// TIA Portal V20 export
DATA_BLOCK "LBP_CtrlEnergy"   // DB1000
TITLE = Ctrl-Energy
{ S7_Optimized_Access := 'FALSE'; DB_Accessible_From_OPC_UA := 'FALSE' }
AUTHOR : SINUMERIK
FAMILY : SINUMERIK_ONE
VERSION : 6.24
// Interface between user program and operating software, contains energy-saving profiles for Ctrl-Energy / Interface entre programme utilisateur et logiciel d'exploitation contient des profils d'économie d'énergie pour Ctrl-Energy
// stored: AutoNumber false, DBAccessibleFromOPCUA false, DBAccessibleFromWebserver false
   VAR RETAIN
      Profile : Array[1..8] of Struct
         ESaveOn { ExternalWritable := 'False'} : Bool;   // Activate energy-saving profile immediately / Activer immédiatement le profil d'économie d'énergie
         ReloadT2 { ExternalWritable := 'False'} : Bool;   // Reload Prewarning time (T2) / Recharger temps de préavis (T2)
         res0_2 { ExternalWritable := 'False'} : Bool;
         res0_3 { ExternalWritable := 'False'} : Bool;
         res0_4 { ExternalWritable := 'False'} : Bool;
         res0_5 { ExternalWritable := 'False'} : Bool;
         res0_6 { ExternalWritable := 'False'} : Bool;
         res0_7 { ExternalWritable := 'False'} : Bool;
         HmiESaveOn : Bool;   // HMI->PLC: Activate energy-saving profile immediately / IHM->AP : activer immédiatement le profil d'économie d'énergie
         res1_1 { ExternalWritable := 'False'} : Bool;
         res1_2 { ExternalWritable := 'False'} : Bool;
         res1_3 { ExternalWritable := 'False'} : Bool;
         res1_4 { ExternalWritable := 'False'} : Bool;
         res1_5 { ExternalWritable := 'False'} : Bool;
         res1_6 { ExternalWritable := 'False'} : Bool;
         res1_7 { ExternalWritable := 'False'} : Bool;
         MasterCompSig { ExternalWritable := 'False'} : Bool;   // Master computer signal / Signal ordinateur maître
         PlcUserSig { ExternalWritable := 'False'} : Bool;   // PLC user signal / AP signal utilisateur
         res2_2 { ExternalWritable := 'False'} : Bool;
         res2_3 { ExternalWritable := 'False'} : Bool;
         res2_4 { ExternalWritable := 'False'} : Bool;
         res2_5 { ExternalWritable := 'False'} : Bool;
         res2_6 { ExternalWritable := 'False'} : Bool;
         res2_7 { ExternalWritable := 'False'} : Bool;
         res3 { ExternalWritable := 'False'} : Byte;
         ESaveIsOn { ExternalWritable := 'False'} : Bool;   // Energy-saving state active / État économie d'énergie actif
         T1Expired { ExternalWritable := 'False'} : Bool;   // Activation time T1 expired / Temps d'activation T1 écoulé
         res4_2 { ExternalWritable := 'False'} : Bool;
         res4_3 { ExternalWritable := 'False'} : Bool;
         res4_4 { ExternalWritable := 'False'} : Bool;
         res4_5 { ExternalWritable := 'False'} : Bool;
         res4_6 { ExternalWritable := 'False'} : Bool;
         res4_7 { ExternalWritable := 'False'} : Bool;
         res5 { ExternalWritable := 'False'} : Byte;
         ActValT1 { ExternalWritable := 'False'} : Int;   // T1 current value / T1 valeur réelle
         ActValT2 { ExternalWritable := 'False'} : Int;   // T2 current value / T2 valeur réelle
         ESaveValid : Bool;   // HMI->PLC: Energy-saving profile valid / IHM->AP : profil d'économie d'énergie valide
         ESaveOff : Bool;   // HMI->PLC: Deactivate energy-saving profileblock energy-saving profile / IHM->AP : désactiver/bloquer le profil d'économie d'énergie
         res10_2 { ExternalWritable := 'False'} : Bool;
         res10_3 { ExternalWritable := 'False'} : Bool;
         res10_4 { ExternalWritable := 'False'} : Bool;
         res10_5 { ExternalWritable := 'False'} : Bool;
         res10_6 { ExternalWritable := 'False'} : Bool;
         res10_7 { ExternalWritable := 'False'} : Bool;
         CondOpPanel : Bool;   // HMI->PLC: Operator panel / IHM->AP : pupitre opérateur
         CondDataTransfer : Bool;   // HMI->PLC: Data transfer / IHM->AP : transmission de données
         CondWindowChange : Bool;   // HMI->PLC: Window change / IHM->AP : changement de fenêtre
         res11_3 { ExternalWritable := 'False'} : Bool;
         res11_4 { ExternalWritable := 'False'} : Bool;
         res11_5 { ExternalWritable := 'False'} : Bool;
         res11_6 { ExternalWritable := 'False'} : Bool;
         res11_7 { ExternalWritable := 'False'} : Bool;
         CondMCP : Bool;   // HMI->PLC: Machine control panel / IHM->AP : pupitre opérateur machine
         res12_1 { ExternalWritable := 'False'} : Bool;
         res12_2 { ExternalWritable := 'False'} : Bool;
         res12_3 { ExternalWritable := 'False'} : Bool;
         res12_4 { ExternalWritable := 'False'} : Bool;
         res12_5 { ExternalWritable := 'False'} : Bool;
         res12_6 { ExternalWritable := 'False'} : Bool;
         res12_7 { ExternalWritable := 'False'} : Bool;
         CondNcChan1 : Bool;   // HMI->PLC: NC channel 1 in reset / IHM->AP : canal CN 1 en Reset
         CondNcChan2 : Bool;   // HMI->PLC: NC channel 2 in reset / IHM->AP : canal CN 2 en Reset
         CondNcChan3 : Bool;   // HMI->PLC: NC channel 3 in reset / IHM->AP : canal CN 3 en Reset
         CondNcChan4 : Bool;   // HMI->PLC: NC channel 4 in reset / IHM->AP : canal CN 4 en Reset
         CondNcChan5 : Bool;   // HMI->PLC: NC channel 5 in reset / IHM->AP : canal CN 5 en Reset
         CondNcChan6 : Bool;   // HMI->PLC: NC channel 6 in reset / IHM->AP : canal CN 6 en Reset
         CondNcChan7 : Bool;   // HMI->PLC: NC channel 7 in reset / IHM->AP : canal CN 7 en Reset
         CondNcChan8 : Bool;   // HMI->PLC: NC channel 8 in reset / IHM->AP : canal CN 8 en Reset
         CondNcChan9 : Bool;   // HMI->PLC: NC channel 9 in reset / IHM->AP : canal CN 9 en Reset
         CondNcChan10 : Bool;   // HMI->PLC: NC channel 10 in reset / IHM->AP : canal CN 10 en Reset
         res14_2 { ExternalWritable := 'False'} : Bool;
         res14_3 { ExternalWritable := 'False'} : Bool;
         res14_4 { ExternalWritable := 'False'} : Bool;
         res14_5 { ExternalWritable := 'False'} : Bool;
         res14_6 { ExternalWritable := 'False'} : Bool;
         res14_7 { ExternalWritable := 'False'} : Bool;
         CondMasterCompSig : Bool;   // HMI->PLC: Master computer signal / IHM->AP : signal ordinateur maître
         CondPlcUserSig : Bool;   // HMI->PLC: PLC user signal / IHM->AP : signal utilisateur AP
         res15_2 { ExternalWritable := 'False'} : Bool;
         res15_3 { ExternalWritable := 'False'} : Bool;
         res15_4 { ExternalWritable := 'False'} : Bool;
         res15_5 { ExternalWritable := 'False'} : Bool;
         res15_6 { ExternalWritable := 'False'} : Bool;
         res15_7 { ExternalWritable := 'False'} : Bool;
         PresetT1 : Int;   // HMI->PLC: Activation time T1 / IHM->AP : temps d'activation T1
         PresetT2 : Int;   // HMI->PLC: Prewarning time T2 / IHM->AP : temps de préavis T2
      END_STRUCT;
   END_VAR
BEGIN
   // Profile[2].ESaveOn : Activate energy-saving profile immediately / Activer immédiatement le profil d'économie d'énergie
   // Profile[3].ESaveOn : Activate energy-saving profile immediately / Activer immédiatement le profil d'économie d'énergie
   // Profile[4].ESaveOn : Activate energy-saving profile immediately / Activer immédiatement le profil d'économie d'énergie
   // Profile[5].ESaveOn : Activate energy-saving profile immediately / Activer immédiatement le profil d'économie d'énergie
   // Profile[6].ESaveOn : Activate energy-saving profile immediately / Activer immédiatement le profil d'économie d'énergie
   // Profile[7].ESaveOn : Activate energy-saving profile immediately / Activer immédiatement le profil d'économie d'énergie
   // Profile[8].ESaveOn : Activate energy-saving profile immediately / Activer immédiatement le profil d'économie d'énergie
   // Profile[2].ReloadT2 : Reload Prewarning time (T2) / Recharger temps de préavis (T2)
   // Profile[3].ReloadT2 : Reload Prewarning time (T2) / Recharger temps de préavis (T2)
   // Profile[4].ReloadT2 : Reload Prewarning time (T2) / Recharger temps de préavis (T2)
   // Profile[5].ReloadT2 : Reload Prewarning time (T2) / Recharger temps de préavis (T2)
   // Profile[6].ReloadT2 : Reload Prewarning time (T2) / Recharger temps de préavis (T2)
   // Profile[7].ReloadT2 : Reload Prewarning time (T2) / Recharger temps de préavis (T2)
   // Profile[8].ReloadT2 : Reload Prewarning time (T2) / Recharger temps de préavis (T2)
   // Profile[2].HmiESaveOn : HMI->PLC: Activate energy-saving profile immediately / IHM->AP : activer immédiatement le profil d'économie d'énergie
   // Profile[3].HmiESaveOn : HMI->PLC: Activate energy-saving profile immediately / IHM->AP : activer immédiatement le profil d'économie d'énergie
   // Profile[4].HmiESaveOn : HMI->PLC: Activate energy-saving profile immediately / IHM->AP : activer immédiatement le profil d'économie d'énergie
   // Profile[5].HmiESaveOn : HMI->PLC: Activate energy-saving profile immediately / IHM->AP : activer immédiatement le profil d'économie d'énergie
   // Profile[6].HmiESaveOn : HMI->PLC: Activate energy-saving profile immediately / IHM->AP : activer immédiatement le profil d'économie d'énergie
   // Profile[7].HmiESaveOn : HMI->PLC: Activate energy-saving profile immediately / IHM->AP : activer immédiatement le profil d'économie d'énergie
   // Profile[8].HmiESaveOn : HMI->PLC: Activate energy-saving profile immediately / IHM->AP : activer immédiatement le profil d'économie d'énergie
   // Profile[2].MasterCompSig : Master computer signal / Signal ordinateur maître
   // Profile[3].MasterCompSig : Master computer signal / Signal ordinateur maître
   // Profile[4].MasterCompSig : Master computer signal / Signal ordinateur maître
   // Profile[5].MasterCompSig : Master computer signal / Signal ordinateur maître
   // Profile[6].MasterCompSig : Master computer signal / Signal ordinateur maître
   // Profile[7].MasterCompSig : Master computer signal / Signal ordinateur maître
   // Profile[8].MasterCompSig : Master computer signal / Signal ordinateur maître
   // Profile[2].PlcUserSig : PLC user signal / AP signal utilisateur
   // Profile[3].PlcUserSig : PLC user signal / AP signal utilisateur
   // Profile[4].PlcUserSig : PLC user signal / AP signal utilisateur
   // Profile[5].PlcUserSig : PLC user signal / AP signal utilisateur
   // Profile[6].PlcUserSig : PLC user signal / AP signal utilisateur
   // Profile[7].PlcUserSig : PLC user signal / AP signal utilisateur
   // Profile[8].PlcUserSig : PLC user signal / AP signal utilisateur
   // Profile[2].ESaveIsOn : Energy-saving state active / État économie d'énergie actif
   // Profile[3].ESaveIsOn : Energy-saving state active / État économie d'énergie actif
   // Profile[4].ESaveIsOn : Energy-saving state active / État économie d'énergie actif
   // Profile[5].ESaveIsOn : Energy-saving state active / État économie d'énergie actif
   // Profile[6].ESaveIsOn : Energy-saving state active / État économie d'énergie actif
   // Profile[7].ESaveIsOn : Energy-saving state active / État économie d'énergie actif
   // Profile[8].ESaveIsOn : Energy-saving state active / État économie d'énergie actif
   // Profile[2].T1Expired : Activation time T1 expired / Temps d'activation T1 écoulé
   // Profile[3].T1Expired : Activation time T1 expired / Temps d'activation T1 écoulé
   // Profile[4].T1Expired : Activation time T1 expired / Temps d'activation T1 écoulé
   // Profile[5].T1Expired : Activation time T1 expired / Temps d'activation T1 écoulé
   // Profile[6].T1Expired : Activation time T1 expired / Temps d'activation T1 écoulé
   // Profile[7].T1Expired : Activation time T1 expired / Temps d'activation T1 écoulé
   // Profile[8].T1Expired : Activation time T1 expired / Temps d'activation T1 écoulé
   // Profile[2].ActValT1 : T1 current value / T1 valeur réelle
   // Profile[3].ActValT1 : T1 current value / T1 valeur réelle
   // Profile[4].ActValT1 : T1 current value / T1 valeur réelle
   // Profile[5].ActValT1 : T1 current value / T1 valeur réelle
   // Profile[6].ActValT1 : T1 current value / T1 valeur réelle
   // Profile[7].ActValT1 : T1 current value / T1 valeur réelle
   // Profile[8].ActValT1 : T1 current value / T1 valeur réelle
   // Profile[2].ActValT2 : T2 current value / T2 valeur réelle
   // Profile[3].ActValT2 : T2 current value / T2 valeur réelle
   // Profile[4].ActValT2 : T2 current value / T2 valeur réelle
   // Profile[5].ActValT2 : T2 current value / T2 valeur réelle
   // Profile[6].ActValT2 : T2 current value / T2 valeur réelle
   // Profile[7].ActValT2 : T2 current value / T2 valeur réelle
   // Profile[8].ActValT2 : T2 current value / T2 valeur réelle
   Profile[1].ESaveValid := TRUE;
   Profile[2].ESaveValid := TRUE;   // HMI->PLC: Energy-saving profile valid / IHM->AP : profil d'économie d'énergie valide
   Profile[3].ESaveValid := TRUE;   // HMI->PLC: Energy-saving profile valid / IHM->AP : profil d'économie d'énergie valide
   // Profile[4].ESaveValid : HMI->PLC: Energy-saving profile valid / IHM->AP : profil d'économie d'énergie valide
   // Profile[5].ESaveValid : HMI->PLC: Energy-saving profile valid / IHM->AP : profil d'économie d'énergie valide
   // Profile[6].ESaveValid : HMI->PLC: Energy-saving profile valid / IHM->AP : profil d'économie d'énergie valide
   // Profile[7].ESaveValid : HMI->PLC: Energy-saving profile valid / IHM->AP : profil d'économie d'énergie valide
   // Profile[8].ESaveValid : HMI->PLC: Energy-saving profile valid / IHM->AP : profil d'économie d'énergie valide
   Profile[1].ESaveOff := TRUE;
   Profile[2].ESaveOff := TRUE;   // HMI->PLC: Deactivate energy-saving profileblock energy-saving profile / IHM->AP : désactiver/bloquer le profil d'économie d'énergie
   Profile[3].ESaveOff := TRUE;   // HMI->PLC: Deactivate energy-saving profileblock energy-saving profile / IHM->AP : désactiver/bloquer le profil d'économie d'énergie
   // Profile[4].ESaveOff : HMI->PLC: Deactivate energy-saving profileblock energy-saving profile / IHM->AP : désactiver/bloquer le profil d'économie d'énergie
   // Profile[5].ESaveOff : HMI->PLC: Deactivate energy-saving profileblock energy-saving profile / IHM->AP : désactiver/bloquer le profil d'économie d'énergie
   // Profile[6].ESaveOff : HMI->PLC: Deactivate energy-saving profileblock energy-saving profile / IHM->AP : désactiver/bloquer le profil d'économie d'énergie
   // Profile[7].ESaveOff : HMI->PLC: Deactivate energy-saving profileblock energy-saving profile / IHM->AP : désactiver/bloquer le profil d'économie d'énergie
   // Profile[8].ESaveOff : HMI->PLC: Deactivate energy-saving profileblock energy-saving profile / IHM->AP : désactiver/bloquer le profil d'économie d'énergie
   // Profile[2].CondOpPanel : HMI->PLC: Operator panel / IHM->AP : pupitre opérateur
   Profile[3].CondOpPanel := TRUE;   // HMI->PLC: Operator panel / IHM->AP : pupitre opérateur
   // Profile[4].CondOpPanel : HMI->PLC: Operator panel / IHM->AP : pupitre opérateur
   // Profile[5].CondOpPanel : HMI->PLC: Operator panel / IHM->AP : pupitre opérateur
   // Profile[6].CondOpPanel : HMI->PLC: Operator panel / IHM->AP : pupitre opérateur
   // Profile[7].CondOpPanel : HMI->PLC: Operator panel / IHM->AP : pupitre opérateur
   // Profile[8].CondOpPanel : HMI->PLC: Operator panel / IHM->AP : pupitre opérateur
   // Profile[2].CondDataTransfer : HMI->PLC: Data transfer / IHM->AP : transmission de données
   Profile[3].CondDataTransfer := TRUE;   // HMI->PLC: Data transfer / IHM->AP : transmission de données
   // Profile[4].CondDataTransfer : HMI->PLC: Data transfer / IHM->AP : transmission de données
   // Profile[5].CondDataTransfer : HMI->PLC: Data transfer / IHM->AP : transmission de données
   // Profile[6].CondDataTransfer : HMI->PLC: Data transfer / IHM->AP : transmission de données
   // Profile[7].CondDataTransfer : HMI->PLC: Data transfer / IHM->AP : transmission de données
   // Profile[8].CondDataTransfer : HMI->PLC: Data transfer / IHM->AP : transmission de données
   // Profile[2].CondWindowChange : HMI->PLC: Window change / IHM->AP : changement de fenêtre
   Profile[3].CondWindowChange := TRUE;   // HMI->PLC: Window change / IHM->AP : changement de fenêtre
   // Profile[4].CondWindowChange : HMI->PLC: Window change / IHM->AP : changement de fenêtre
   // Profile[5].CondWindowChange : HMI->PLC: Window change / IHM->AP : changement de fenêtre
   // Profile[6].CondWindowChange : HMI->PLC: Window change / IHM->AP : changement de fenêtre
   // Profile[7].CondWindowChange : HMI->PLC: Window change / IHM->AP : changement de fenêtre
   // Profile[8].CondWindowChange : HMI->PLC: Window change / IHM->AP : changement de fenêtre
   Profile[2].CondMCP := TRUE;   // HMI->PLC: Machine control panel / IHM->AP : pupitre opérateur machine
   Profile[3].CondMCP := TRUE;   // HMI->PLC: Machine control panel / IHM->AP : pupitre opérateur machine
   // Profile[4].CondMCP : HMI->PLC: Machine control panel / IHM->AP : pupitre opérateur machine
   // Profile[5].CondMCP : HMI->PLC: Machine control panel / IHM->AP : pupitre opérateur machine
   // Profile[6].CondMCP : HMI->PLC: Machine control panel / IHM->AP : pupitre opérateur machine
   // Profile[7].CondMCP : HMI->PLC: Machine control panel / IHM->AP : pupitre opérateur machine
   // Profile[8].CondMCP : HMI->PLC: Machine control panel / IHM->AP : pupitre opérateur machine
   Profile[1].CondNcChan1 := TRUE;
   Profile[2].CondNcChan1 := TRUE;   // HMI->PLC: NC channel 1 in reset / IHM->AP : canal CN 1 en Reset
   Profile[3].CondNcChan1 := TRUE;   // HMI->PLC: NC channel 1 in reset / IHM->AP : canal CN 1 en Reset
   // Profile[4].CondNcChan1 : HMI->PLC: NC channel 1 in reset / IHM->AP : canal CN 1 en Reset
   // Profile[5].CondNcChan1 : HMI->PLC: NC channel 1 in reset / IHM->AP : canal CN 1 en Reset
   // Profile[6].CondNcChan1 : HMI->PLC: NC channel 1 in reset / IHM->AP : canal CN 1 en Reset
   // Profile[7].CondNcChan1 : HMI->PLC: NC channel 1 in reset / IHM->AP : canal CN 1 en Reset
   // Profile[8].CondNcChan1 : HMI->PLC: NC channel 1 in reset / IHM->AP : canal CN 1 en Reset
   Profile[1].CondNcChan2 := TRUE;
   Profile[2].CondNcChan2 := TRUE;   // HMI->PLC: NC channel 2 in reset / IHM->AP : canal CN 2 en Reset
   Profile[3].CondNcChan2 := TRUE;   // HMI->PLC: NC channel 2 in reset / IHM->AP : canal CN 2 en Reset
   // Profile[4].CondNcChan2 : HMI->PLC: NC channel 2 in reset / IHM->AP : canal CN 2 en Reset
   // Profile[5].CondNcChan2 : HMI->PLC: NC channel 2 in reset / IHM->AP : canal CN 2 en Reset
   // Profile[6].CondNcChan2 : HMI->PLC: NC channel 2 in reset / IHM->AP : canal CN 2 en Reset
   // Profile[7].CondNcChan2 : HMI->PLC: NC channel 2 in reset / IHM->AP : canal CN 2 en Reset
   // Profile[8].CondNcChan2 : HMI->PLC: NC channel 2 in reset / IHM->AP : canal CN 2 en Reset
   Profile[1].CondNcChan3 := TRUE;
   Profile[2].CondNcChan3 := TRUE;   // HMI->PLC: NC channel 3 in reset / IHM->AP : canal CN 3 en Reset
   Profile[3].CondNcChan3 := TRUE;   // HMI->PLC: NC channel 3 in reset / IHM->AP : canal CN 3 en Reset
   // Profile[4].CondNcChan3 : HMI->PLC: NC channel 3 in reset / IHM->AP : canal CN 3 en Reset
   // Profile[5].CondNcChan3 : HMI->PLC: NC channel 3 in reset / IHM->AP : canal CN 3 en Reset
   // Profile[6].CondNcChan3 : HMI->PLC: NC channel 3 in reset / IHM->AP : canal CN 3 en Reset
   // Profile[7].CondNcChan3 : HMI->PLC: NC channel 3 in reset / IHM->AP : canal CN 3 en Reset
   // Profile[8].CondNcChan3 : HMI->PLC: NC channel 3 in reset / IHM->AP : canal CN 3 en Reset
   Profile[1].CondNcChan4 := TRUE;
   Profile[2].CondNcChan4 := TRUE;   // HMI->PLC: NC channel 4 in reset / IHM->AP : canal CN 4 en Reset
   Profile[3].CondNcChan4 := TRUE;   // HMI->PLC: NC channel 4 in reset / IHM->AP : canal CN 4 en Reset
   // Profile[4].CondNcChan4 : HMI->PLC: NC channel 4 in reset / IHM->AP : canal CN 4 en Reset
   // Profile[5].CondNcChan4 : HMI->PLC: NC channel 4 in reset / IHM->AP : canal CN 4 en Reset
   // Profile[6].CondNcChan4 : HMI->PLC: NC channel 4 in reset / IHM->AP : canal CN 4 en Reset
   // Profile[7].CondNcChan4 : HMI->PLC: NC channel 4 in reset / IHM->AP : canal CN 4 en Reset
   // Profile[8].CondNcChan4 : HMI->PLC: NC channel 4 in reset / IHM->AP : canal CN 4 en Reset
   Profile[1].CondNcChan5 := TRUE;
   Profile[2].CondNcChan5 := TRUE;   // HMI->PLC: NC channel 5 in reset / IHM->AP : canal CN 5 en Reset
   Profile[3].CondNcChan5 := TRUE;   // HMI->PLC: NC channel 5 in reset / IHM->AP : canal CN 5 en Reset
   // Profile[4].CondNcChan5 : HMI->PLC: NC channel 5 in reset / IHM->AP : canal CN 5 en Reset
   // Profile[5].CondNcChan5 : HMI->PLC: NC channel 5 in reset / IHM->AP : canal CN 5 en Reset
   // Profile[6].CondNcChan5 : HMI->PLC: NC channel 5 in reset / IHM->AP : canal CN 5 en Reset
   // Profile[7].CondNcChan5 : HMI->PLC: NC channel 5 in reset / IHM->AP : canal CN 5 en Reset
   // Profile[8].CondNcChan5 : HMI->PLC: NC channel 5 in reset / IHM->AP : canal CN 5 en Reset
   Profile[1].CondNcChan6 := TRUE;
   Profile[2].CondNcChan6 := TRUE;   // HMI->PLC: NC channel 6 in reset / IHM->AP : canal CN 6 en Reset
   Profile[3].CondNcChan6 := TRUE;   // HMI->PLC: NC channel 6 in reset / IHM->AP : canal CN 6 en Reset
   // Profile[4].CondNcChan6 : HMI->PLC: NC channel 6 in reset / IHM->AP : canal CN 6 en Reset
   // Profile[5].CondNcChan6 : HMI->PLC: NC channel 6 in reset / IHM->AP : canal CN 6 en Reset
   // Profile[6].CondNcChan6 : HMI->PLC: NC channel 6 in reset / IHM->AP : canal CN 6 en Reset
   // Profile[7].CondNcChan6 : HMI->PLC: NC channel 6 in reset / IHM->AP : canal CN 6 en Reset
   // Profile[8].CondNcChan6 : HMI->PLC: NC channel 6 in reset / IHM->AP : canal CN 6 en Reset
   Profile[1].CondNcChan7 := TRUE;
   Profile[2].CondNcChan7 := TRUE;   // HMI->PLC: NC channel 7 in reset / IHM->AP : canal CN 7 en Reset
   Profile[3].CondNcChan7 := TRUE;   // HMI->PLC: NC channel 7 in reset / IHM->AP : canal CN 7 en Reset
   // Profile[4].CondNcChan7 : HMI->PLC: NC channel 7 in reset / IHM->AP : canal CN 7 en Reset
   // Profile[5].CondNcChan7 : HMI->PLC: NC channel 7 in reset / IHM->AP : canal CN 7 en Reset
   // Profile[6].CondNcChan7 : HMI->PLC: NC channel 7 in reset / IHM->AP : canal CN 7 en Reset
   // Profile[7].CondNcChan7 : HMI->PLC: NC channel 7 in reset / IHM->AP : canal CN 7 en Reset
   // Profile[8].CondNcChan7 : HMI->PLC: NC channel 7 in reset / IHM->AP : canal CN 7 en Reset
   Profile[1].CondNcChan8 := TRUE;
   Profile[2].CondNcChan8 := TRUE;   // HMI->PLC: NC channel 8 in reset / IHM->AP : canal CN 8 en Reset
   Profile[3].CondNcChan8 := TRUE;   // HMI->PLC: NC channel 8 in reset / IHM->AP : canal CN 8 en Reset
   // Profile[4].CondNcChan8 : HMI->PLC: NC channel 8 in reset / IHM->AP : canal CN 8 en Reset
   // Profile[5].CondNcChan8 : HMI->PLC: NC channel 8 in reset / IHM->AP : canal CN 8 en Reset
   // Profile[6].CondNcChan8 : HMI->PLC: NC channel 8 in reset / IHM->AP : canal CN 8 en Reset
   // Profile[7].CondNcChan8 : HMI->PLC: NC channel 8 in reset / IHM->AP : canal CN 8 en Reset
   // Profile[8].CondNcChan8 : HMI->PLC: NC channel 8 in reset / IHM->AP : canal CN 8 en Reset
   Profile[1].CondNcChan9 := TRUE;
   Profile[2].CondNcChan9 := TRUE;   // HMI->PLC: NC channel 9 in reset / IHM->AP : canal CN 9 en Reset
   Profile[3].CondNcChan9 := TRUE;   // HMI->PLC: NC channel 9 in reset / IHM->AP : canal CN 9 en Reset
   // Profile[4].CondNcChan9 : HMI->PLC: NC channel 9 in reset / IHM->AP : canal CN 9 en Reset
   // Profile[5].CondNcChan9 : HMI->PLC: NC channel 9 in reset / IHM->AP : canal CN 9 en Reset
   // Profile[6].CondNcChan9 : HMI->PLC: NC channel 9 in reset / IHM->AP : canal CN 9 en Reset
   // Profile[7].CondNcChan9 : HMI->PLC: NC channel 9 in reset / IHM->AP : canal CN 9 en Reset
   // Profile[8].CondNcChan9 : HMI->PLC: NC channel 9 in reset / IHM->AP : canal CN 9 en Reset
   Profile[1].CondNcChan10 := TRUE;
   Profile[2].CondNcChan10 := TRUE;   // HMI->PLC: NC channel 10 in reset / IHM->AP : canal CN 10 en Reset
   Profile[3].CondNcChan10 := TRUE;   // HMI->PLC: NC channel 10 in reset / IHM->AP : canal CN 10 en Reset
   // Profile[4].CondNcChan10 : HMI->PLC: NC channel 10 in reset / IHM->AP : canal CN 10 en Reset
   // Profile[5].CondNcChan10 : HMI->PLC: NC channel 10 in reset / IHM->AP : canal CN 10 en Reset
   // Profile[6].CondNcChan10 : HMI->PLC: NC channel 10 in reset / IHM->AP : canal CN 10 en Reset
   // Profile[7].CondNcChan10 : HMI->PLC: NC channel 10 in reset / IHM->AP : canal CN 10 en Reset
   // Profile[8].CondNcChan10 : HMI->PLC: NC channel 10 in reset / IHM->AP : canal CN 10 en Reset
   // Profile[2].CondMasterCompSig : HMI->PLC: Master computer signal / IHM->AP : signal ordinateur maître
   // Profile[3].CondMasterCompSig : HMI->PLC: Master computer signal / IHM->AP : signal ordinateur maître
   // Profile[4].CondMasterCompSig : HMI->PLC: Master computer signal / IHM->AP : signal ordinateur maître
   // Profile[5].CondMasterCompSig : HMI->PLC: Master computer signal / IHM->AP : signal ordinateur maître
   // Profile[6].CondMasterCompSig : HMI->PLC: Master computer signal / IHM->AP : signal ordinateur maître
   // Profile[7].CondMasterCompSig : HMI->PLC: Master computer signal / IHM->AP : signal ordinateur maître
   // Profile[8].CondMasterCompSig : HMI->PLC: Master computer signal / IHM->AP : signal ordinateur maître
   Profile[1].CondPlcUserSig := TRUE;
   Profile[2].CondPlcUserSig := TRUE;   // HMI->PLC: PLC user signal / IHM->AP : signal utilisateur AP
   Profile[3].CondPlcUserSig := TRUE;   // HMI->PLC: PLC user signal / IHM->AP : signal utilisateur AP
   // Profile[4].CondPlcUserSig : HMI->PLC: PLC user signal / IHM->AP : signal utilisateur AP
   // Profile[5].CondPlcUserSig : HMI->PLC: PLC user signal / IHM->AP : signal utilisateur AP
   // Profile[6].CondPlcUserSig : HMI->PLC: PLC user signal / IHM->AP : signal utilisateur AP
   // Profile[7].CondPlcUserSig : HMI->PLC: PLC user signal / IHM->AP : signal utilisateur AP
   // Profile[8].CondPlcUserSig : HMI->PLC: PLC user signal / IHM->AP : signal utilisateur AP
   Profile[1].PresetT1 := 60;
   Profile[2].PresetT1 := 120;   // HMI->PLC: Activation time T1 / IHM->AP : temps d'activation T1
   Profile[3].PresetT1 := 600;   // HMI->PLC: Activation time T1 / IHM->AP : temps d'activation T1
   // Profile[4].PresetT1 : HMI->PLC: Activation time T1 / IHM->AP : temps d'activation T1
   // Profile[5].PresetT1 : HMI->PLC: Activation time T1 / IHM->AP : temps d'activation T1
   // Profile[6].PresetT1 : HMI->PLC: Activation time T1 / IHM->AP : temps d'activation T1
   // Profile[7].PresetT1 : HMI->PLC: Activation time T1 / IHM->AP : temps d'activation T1
   // Profile[8].PresetT1 : HMI->PLC: Activation time T1 / IHM->AP : temps d'activation T1
   Profile[1].PresetT2 := 120;
   Profile[2].PresetT2 := 300;   // HMI->PLC: Prewarning time T2 / IHM->AP : temps de préavis T2
   // Profile[3].PresetT2 : HMI->PLC: Prewarning time T2 / IHM->AP : temps de préavis T2
   // Profile[4].PresetT2 : HMI->PLC: Prewarning time T2 / IHM->AP : temps de préavis T2
   // Profile[5].PresetT2 : HMI->PLC: Prewarning time T2 / IHM->AP : temps de préavis T2
   // Profile[6].PresetT2 : HMI->PLC: Prewarning time T2 / IHM->AP : temps de préavis T2
   // Profile[7].PresetT2 : HMI->PLC: Prewarning time T2 / IHM->AP : temps de préavis T2
   // Profile[8].PresetT2 : HMI->PLC: Prewarning time T2 / IHM->AP : temps de préavis T2
END_DATA_BLOCK
